TYPE DUT_MotionStageNCParams :
STRUCT
    // NC Forward Limit Switch: TRUE if ok to move
    {attribute 'pytmc' := '
        pv: FEncOffset
        io: i
        field: ZNAM FALSE
        field: ONAM TRUE
        field: DESC FALSE if forward limit hit
    '}
    fEncOffset AT %I*: LREAL;
    // NC Backward Limit Switch: TRUE if ok to move
    {attribute 'pytmc' := '
        pv: fEncScaleFactor
        io: i
        field: ZNAM FALSE
        field: ONAM TRUE
        field: DESC FALSE if reverse limit hit
    '}
    fEncScaleFactor AT %I*: LREAL;
    //test
END_STRUCT
END_TYPE

(* stored: Version 1.1.0.1, ProductVersion 3.1.4022.18
   DUT DUT_MotionStageNCParams: Id {b38ca476-dbb9-4b4a-a811-68bc4bdb9b25} *)
